(* Schneider Machine Expert - Basic project envio binario 16, file version 2.7.0.0 *)
(* ProjectInformations: Name=New project *)

HARDWARE
  Cpu 0: TM221ME16T/G
  ModuleExtensionObject 0: TM3DI16/G
  EthernetConfiguration: NetworkName=M221, IpAllocationMode=FixedAddress, IpAddress=192.168.127.130, SubnetMask=255.255.255.0
  SerialLineConfiguration: Baud=Baud19200, Parity=ParityEven, DataBits=DataBits8, StopBits=StopBits1, PhysicalMedium=PhysicalMediumRs485, TransmissionMode=TransmissionModeModbusRtu, SlaveId=1, Addressing=SlaveAddressing
  MastTask: UsePeriodScanMode=false, PeriodScan=100
  FastTask: Period=255
  CpuBehavior: StartingMode=StartAsPreviousState, AutoSaveRamOnEeprom=true, WatchdogPeriod=250

SYMBOLS  (address, symbol, comment, settings)
  %M0       BIT1
  %M1       BIT2
  %M2       BIT3
  %M3       BIT4
  %M4       BIT5
  %M5       BIT6
  %M6       BIT7
  %M7       BIT8
  %M8       BIT9
  %M9       BIT10
  %M10      BIT11
  %M11      BIT12
  %M12      BIT13
  %M13      BIT14
  %M14      BIT15
  %M15      BIT16

POU New POU
  (* SectionNumber=1 *)

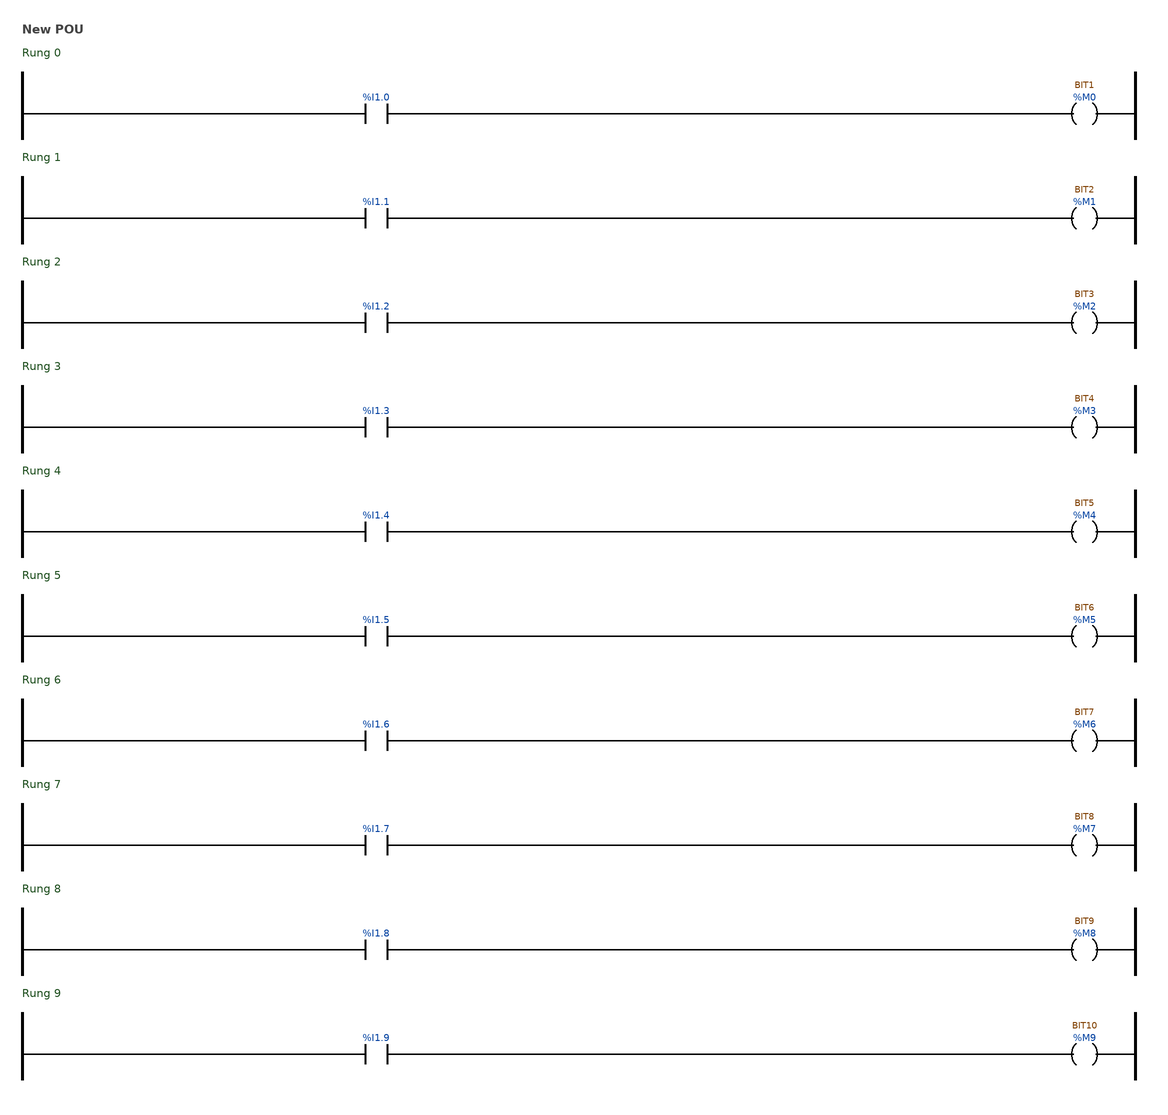

// Rung 0
  LD %I1.0
  ST %M0                  (* BIT1 *)
  // as ST:
  //   BIT1 := %I1.0;

// Rung 1
  LD %I1.1
  ST %M1                  (* BIT2 *)
  // as ST:
  //   BIT2 := %I1.1;

// Rung 2
  LD %I1.2
  ST %M2                  (* BIT3 *)
  // as ST:
  //   BIT3 := %I1.2;

// Rung 3
  LD %I1.3
  ST %M3                  (* BIT4 *)
  // as ST:
  //   BIT4 := %I1.3;

// Rung 4
  LD %I1.4
  ST %M4                  (* BIT5 *)
  // as ST:
  //   BIT5 := %I1.4;

// Rung 5
  LD %I1.5
  ST %M5                  (* BIT6 *)
  // as ST:
  //   BIT6 := %I1.5;

// Rung 6
  LD %I1.6
  ST %M6                  (* BIT7 *)
  // as ST:
  //   BIT7 := %I1.6;

// Rung 7
  LD %I1.7
  ST %M7                  (* BIT8 *)
  // as ST:
  //   BIT8 := %I1.7;

// Rung 8
  LD %I1.8
  ST %M8                  (* BIT9 *)
  // as ST:
  //   BIT9 := %I1.8;

// Rung 9
  LD %I1.9
  ST %M9                  (* BIT10 *)
  // as ST:
  //   BIT10 := %I1.9;

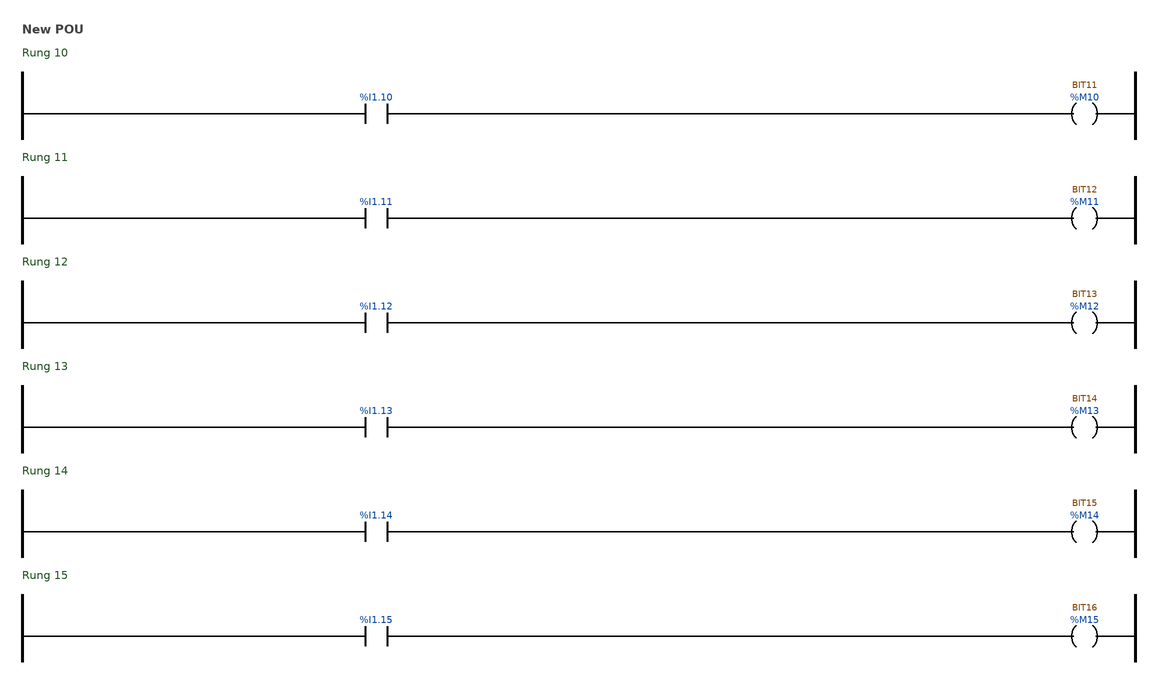

// Rung 10
  LD %I1.10
  ST %M10                 (* BIT11 *)
  // as ST:
  //   BIT11 := %I1.10;

// Rung 11
  LD %I1.11
  ST %M11                 (* BIT12 *)
  // as ST:
  //   BIT12 := %I1.11;

// Rung 12
  LD %I1.12
  ST %M12                 (* BIT13 *)
  // as ST:
  //   BIT13 := %I1.12;

// Rung 13
  LD %I1.13
  ST %M13                 (* BIT14 *)
  // as ST:
  //   BIT14 := %I1.13;

// Rung 14
  LD %I1.14
  ST %M14                 (* BIT15 *)
  // as ST:
  //   BIT15 := %I1.14;

// Rung 15
  LD %I1.15
  ST %M15                 (* BIT16 *)
  // as ST:
  //   BIT16 := %I1.15;
